// TwinCAT 3 PLC project PLC_Tank
// ProgramVersion: 3.1.4024.0
// libraries:
//   Tc2_ControllerToolbox, * (Beckhoff Automation GmbH)
//   Tc2_ModbusSrv, * (Beckhoff Automation GmbH)
//   Tc2_Standard, * (Beckhoff Automation GmbH)
//   Tc2_System, * (Beckhoff Automation GmbH)
//   Tc3_Module, * (Beckhoff Automation GmbH)
//   VisuDialogs, * (System)
//   VisuSymbols,3.5.10.0,System
// project tree:
//   DUTs/ TAnalogConversion.TcDUT (not stored), TEngine.TcDUT (not stored), TEngineCmd.TcDUT (not stored), THeaterState.TcDUT (not stored), THeaterCmd.TcDUT (not stored), THeater.TcDUT (not stored), TPhaseHeating.TcDUT (not stored), TPhaseCmd.TcDUT (not stored), TPhaseDraining.TcDUT (not stored), TPhaseFilling.TcDUT (not stored), TPhaseMixing.TcDUT (not stored), TPhaseState.TcDUT (not stored), TValveState.TcDUT (not stored), TValveCmd.TcDUT (not stored), TEngineState.TcDUT (not stored), TTank.TcDUT (not stored), TValve.TcDUT (not stored)
//   / GlobalTextList.TcGTLO, PlcTask.TcTTO (not stored), PlcTask500ms.TcTTO (not stored), Visualization Manager.TcVMO (not stored)
//   GVLs/ Global.TcGVL
//   POUs/ Draining.TcPOU, Engine_1DO.TcPOU, FB_Tank.TcPOU (not stored), Filling.TcPOU, Heater.TcPOU, Heating.TcPOU, Main_Batch.TcPOU (not stored), MB_Connector.TcPOU, Mixing.TcPOU, Test.TcPOU (not stored), Valve_2DO.TcPOU, MAIN.TcPOU
//   POUs/Misc/ EngToRaw.TcPOU (not stored), RawToEng.TcPOU (not stored), XNOR.TcPOU
//   VISUs/ Visualization.TcVIS
// real-time tasks:
//   TASK PlcTask: cycle T#100000us, priority 20, ADS port 350
//   TASK PlcTask500ms: cycle T#500ms, priority 1, ADS port 351

// ---- GVLs/Global.TcGVL
{attribute 'qualified_only'}
VAR_GLOBAL
	Tank1 : TTank;
	

	secImp : BOOL;
	
	diMixerRun: BOOL;
	diMixerError : BOOL;
	diValveFillOpen : BOOL;
	diValveFillClose : BOOL;
	diValveFillError : BOOL;
	diValveDrainOpen : BOOL;
	diValveDrainClose : BOOL;
	diValveDrainError : BOOL;
	
	aiWaterLevel : WORD;
	aiWaterTemp : WORD;
	
	doMixerStart : BOOL;
	doValveFillOpen : BOOL;
	doValveFillClose : BOOL;
	doValveDrainOpen : BOOL;
	doValveDrainClose : BOOL;
	doHeatingEnable : BOOL;
	
	aoReqPowerOfHeating : WORD;

END_VAR

VAR_GLOBAL CONSTANT
	Running : INT := 0;
	Stop : INT := 1;
	RunningAndError : INT := 2;
	Err : INT := 3;

	PhIdle : INT := 0;
	PhRunning : INT := 1;
	PhPause : INT := 2;
	
    Open : INT := 0;
	Closed : INT := 1;
	OpenAndErr : INT := 2;
	ClosedAndErr : INT := 3;
	NotOpenNotClosedNotErr : INT := 4;
	NotOpenNotClosedAndErr : INT := 5;
	OpenAndClosedAndErr : INT := 6;
	OpenAndClosedNotErr : INT := 7;
END_VAR

// ---- POUs/Draining.TcPOU
FUNCTION_BLOCK Draining
VAR_INPUT
	diEnabled : BOOL;
END_VAR
VAR_OUTPUT
	doEnabled : BOOL;
END_VAR
VAR_IN_OUT
	DrainingPhase : TPhaseDraining;
	DrainingValve : TValve;
	
END_VAR
VAR
	State_temp	:	INT :=0;
END_VAR

{region "Aut/Man"}
    // switching state of engine - automatic or manual control (default state is manual)
		IF	DrainingPhase.Cmd.ManCtrl	THEN
		DrainingPhase.State.ManCtrl	:= TRUE;
		DrainingPhase.State.AutCtrl := FALSE;			 
	END_IF	 
  
	IF	DrainingPhase.Cmd.AutCtrl	THEN
		DrainingPhase.State.ManCtrl	:= FALSE;
		DrainingPhase.State.AutCtrl := TRUE;			 
	END_IF
		 
	IF	(DrainingPhase.Cmd.ManCtrl AND DrainingPhase.Cmd.AutCtrl) 	THEN
		DrainingPhase.State.ManCtrl	:= TRUE;
		DrainingPhase.State.AutCtrl := FALSE;		 
	END_IF
	
	DrainingPhase.Cmd.ManCtrl	:= FALSE;
	DrainingPhase.Cmd.AutCtrl	:= FALSE;	 
	

{endregion}

{region "ManCtrl"}
    // processing manual actions - if command is processed, it is sets to FALSE even if can't be processed
    // Phase commands are start, stop, pause and resume 
    // Start - open draining valve 
    // Stop - close draining valve
    // Pause - close draining valve
    // Resume - open draining valve
    // real states of phase are writed into states in phase structure
  	IF	DrainingPhase.State.ManCtrl	THEN
			 
	CASE State_temp OF
	
	0:	//IDLE STATE - nothing happens
		 DrainingPhase.State.Running	:= FALSE;
		 DrainingPhase.State.Paused	:= FALSE;
		 DrainingPhase.State.Idle	:= TRUE;
		 IF DrainingPhase.Cmd.StartMan THEN
				  State_temp	:= 1;
			  END_IF
	1:	//RUNNING STATE - manual running
		 DrainingPhase.State.Running	:= TRUE;
		 DrainingPhase.State.Paused	:= FALSE;
		 DrainingPhase.State.Idle	:= FALSE;
		 IF DrainingPhase.Cmd.StopMan THEN
				  State_temp	:= 0;
		 ELSIF DrainingPhase.Cmd.PauseMan THEN
				  State_temp := 2;	
		 	 END_IF
	2:	//PAUSED STATE - in PAUSE you are able to go into either RUNNING or IDLE
		 DrainingPhase.State.Running	:= FALSE;
		 DrainingPhase.State.Paused	:= TRUE;
		 DrainingPhase.State.Idle	:= FALSE;
		IF DrainingPhase.Cmd.ResumeMan THEN
				  State_temp	:= 1;
		 ELSIF DrainingPhase.Cmd.StopMan THEN
				  State_temp := 0;	
		 	END_IF
				  
	END_CASE
		
	DrainingPhase.Cmd.StartMan	:= FALSE; 
	DrainingPhase.Cmd.PauseMan	:= FALSE;
	DrainingPhase.Cmd.StopMan	:= FALSE;
	DrainingPhase.Cmd.ResumeMan	:= FALSE;
   END_IF
	   
{endregion}

{region "AutCtrl"}
    //if request to run in automatic mode -> set auto request to open of filling valve to 1 and close to 0, if not open 0 close 1
    // commands should be sets to false after their processing
	 IF DrainingPhase.State.AutCtrl	THEN
		
	IF	DrainingPhase.Cmd.StartAut THEN
		DrainingPhase.State.Running	:= TRUE;
		DrainingPhase.State.Idle		:= FALSE;	 
	ELSIF	DrainingPhase.Cmd.StopAut THEN	
		DrainingPhase.State.Idle		:= TRUE;
		DrainingPhase.State.Running	:= FALSE;
	END_IF

	DrainingPhase.Cmd.StartAut	:= FALSE;
	DrainingPhase.Cmd.StopAut	:= FALSE;	
   
  END_IF
	
   
{endregion}
{region "Done"}
    //every phase should have finish condition - draining phase - if water level is below requested level
    //after that done state should be setted to 1
   DrainingPhase.ParamDrainLevel	:= 0.02;		//temporary inicialization for testing
		
	IF	DrainingPhase.ParamDrainLevel >= Global.Tank1.Filling.WaterLevel	THEN	//just for now I am using variablbe from Filling	
		DrainingPhase.Cmd.StopMan	:= TRUE;										//perhaps I gotta create new FB EngToRaw for Draining.WaterLevel
		DrainingPhase.Cmd.StopAut	:= TRUE;
		DrainingPhase.State.Done		:= TRUE;		
	ELSIF	DrainingPhase.Cmd.ResetDone THEN
		DrainingPhase.State.Done	:= FALSE;
		DrainingPhase.Cmd.ResetDone := FALSE;
	ELSE
		DrainingPhase.State.Done	:= FALSE;
    END_IF
{endregion}

{region "States"} 
    //Command valve in cases of states
	IF DrainingPhase.State.Running  AND NOT DrainingPhase.State.Idle AND NOT DrainingPhase.State.Paused AND NOT DrainingPhase.State.Done THEN 
        DrainingValve.Cmd.Req2OpenAut := TRUE;
        DrainingValve.Cmd.Req2CloseAut := FALSE;
    ELSE
        DrainingValve.Cmd.Req2OpenAut := FALSE;
        DrainingValve.Cmd.Req2CloseAut := TRUE;
    END_IF;

   
{endregion}

// delault state of phase - if not any state sets state to idle
IF (NOT DrainingPhase.State.Idle) AND (NOT DrainingPhase.State.Paused) AND (NOT DrainingPhase.State.Running) THEN
    DrainingPhase.State.Idle := 1;
END_IF;

// write binary states into int value for visualization
IF DrainingPhase.State.Idle THEN
    DrainingPhase.State.StateInt := Global.PhIdle;
ELSIF DrainingPhase.State.Running THEN
    DrainingPhase.State.StateInt := Global.PhRunning;
ELSE
    DrainingPhase.State.StateInt := Global.PhPause;
END_IF;

//Ponechte pro moznost retezeni volani bloku v LAD
doEnabled := diEnabled;

END_FUNCTION_BLOCK

// ---- POUs/Filling.TcPOU
FUNCTION_BLOCK Filling
VAR_INPUT
	diEnabled : BOOL;
END_VAR
VAR_OUTPUT
	doEnabled : BOOL;
END_VAR
VAR_IN_OUT
	FillingPhase : TPhaseFilling;
	FillingValve : TValve;
END_VAR
VAR
	State_temp	: INT := 0;
END_VAR

{region "REGION Aut/Man"}
    // switching state of engine - automatic or manual control (default state is manual)
	IF	FillingPhase.Cmd.ManCtrl	THEN
		FillingPhase.State.ManCtrl	:= TRUE;
		FillingPhase.State.AutCtrl	:= FALSE;			 
	END_IF	 
  
	IF	FillingPhase.Cmd.AutCtrl	THEN
		FillingPhase.State.ManCtrl	:= FALSE;
		FillingPhase.State.AutCtrl	:= TRUE;			 
	END_IF
		 
	IF	(FillingPhase.Cmd.ManCtrl AND FillingPhase.Cmd.AutCtrl) 	THEN
		FillingPhase.State.ManCtrl	:= TRUE;
		FillingPhase.State.AutCtrl	:= FALSE;			 
	END_IF
	   
	FillingPhase.Cmd.AutCtrl := FALSE;
	FillingPhase.Cmd.ManCtrl := FALSE;
{endregion}

{region "ManCtrl"}
    // processing manual actions - if command is processed, it is sets to FALSE even if can't be processed
    // Phase commands are start, stop, pause and resume 
    // Start - open filling valve 
    // Stop - close filling valve
    // Pause - close filling valve
    // Resume - open filling valve
    // real states of phase are writed into states in phase structure
	
	IF	FillingPhase.State.ManCtrl	THEN
			 
	CASE State_temp OF
	
	0:	//IDLE STATE - nothing happens
		 FillingPhase.State.Running	:= FALSE;
		 FillingPhase.State.Paused	:= FALSE;
		 FillingPhase.State.Idle	:= TRUE;
		 IF FillingPhase.Cmd.StartMan THEN
				  State_temp	:= 1;
			  END_IF
	1:	//RUNNING STATE - manual running
		 FillingPhase.State.Running	:= TRUE;
		 FillingPhase.State.Paused	:= FALSE;
		 FillingPhase.State.Idle	:= FALSE;
		 IF FillingPhase.Cmd.StopMan THEN
				  State_temp	:= 0;
		 ELSIF FillingPhase.Cmd.PauseMan THEN
				  State_temp := 2;	
		 	 END_IF
	2:	//PAUSED STATE - in PAUSE you are able to go into either RUNNING or IDLE
		 FillingPhase.State.Running	:= FALSE;
		 FillingPhase.State.Paused	:= TRUE;
		 FillingPhase.State.Idle	:= FALSE;
		IF FillingPhase.Cmd.ResumeMan THEN
				  State_temp	:= 1;
		 ELSIF FillingPhase.Cmd.StopMan THEN
				  State_temp := 0;	
		 	END_IF
				  
	END_CASE
		
	FillingPhase.Cmd.StartMan	:= FALSE; 
	FillingPhase.Cmd.PauseMan	:= FALSE;
	FillingPhase.Cmd.StopMan	:= FALSE;
	FillingPhase.Cmd.ResumeMan	:= FALSE;
   END_IF
{endregion}

{region "AutCtrl"}
    // if request to run in automatic mode and phase can be run in automatic mode switch phase to running
  IF FillingPhase.State.AutCtrl	THEN
		
	IF	FillingPhase.Cmd.StartAut THEN
		FillingPhase.State.Running	:= TRUE;
		FillingPhase.State.Idle		:= FALSE;	 
	ELSIF	FillingPhase.Cmd.StopAut THEN	
		FillingPhase.State.Idle		:= TRUE;
		FillingPhase.State.Running	:= FALSE;
	END_IF

	FillingPhase.Cmd.StartAut	:= FALSE;
	FillingPhase.Cmd.StopAut	:= FALSE;	
   
  END_IF
			 
   
{endregion}

{region "Done"}
    //every phase should have finish condition - filling phase - if water level is above requested level
    //after that done state should be setted to 1
	FillingPhase.ParamFillLevel	:= 1.5;		//temporary inicialization for testing
		 
	IF	FillingPhase.ParamFillLevel <= FillingPhase.WaterLevel	THEN
		FillingPhase.Cmd.StopMan	:= TRUE;
		FillingPhase.Cmd.StopAut	:= TRUE;
		FillingPhase.State.Done		:= TRUE;		
	ELSIF	FillingPhase.Cmd.ResetDone THEN
		FillingPhase.State.Done	:= FALSE;
		FillingPhase.Cmd.ResetDone := FALSE;
    END_IF
{endregion}

{region "States"} 
    //Command valve in cases of states
	IF FillingPhase.State.Running  AND NOT FillingPhase.State.Idle AND NOT FillingPhase.State.Paused AND NOT FillingPhase.State.Done THEN 
        FillingValve.Cmd.Req2OpenAut := TRUE;
		FillingValve.Cmd.Req2CloseAut := FALSE;			 
    ELSE
        FillingValve.Cmd.Req2OpenAut := FALSE;
        FillingValve.Cmd.Req2CloseAut := TRUE;
    END_IF;

{endregion}


// delault state of phase - if not any state sets state to idle
IF NOT FillingPhase.State.Idle AND NOT FillingPhase.State.Paused AND NOT FillingPhase.State.Running THEN
    FillingPhase.State.Idle := 1;
END_IF;

// write binary states into int value for visualization
IF FillingPhase.State.Idle THEN
    FillingPhase.State.Stateint := Global.PhIdle;
ELSIF FillingPhase.State.Running THEN
    FillingPhase.State.Stateint := Global.PhRunning;
ELSE
    FillingPhase.State.Stateint := Global.PhPause;
END_IF;

// Ponechte pro moznost retezeni volani bloku v LAD
doEnabled := diEnabled;

END_FUNCTION_BLOCK

// ---- POUs/Engine_1DO.TcPOU
FUNCTION_BLOCK Engine_1DO
VAR_INPUT
	iRunning : BOOL;
	iError : BOOL;
	iSecImp : BOOL;
END_VAR
VAR_OUTPUT
	oRun : BOOL;
END_VAR
VAR_IN_OUT
	ioEngStruct : TEngine;
END_VAR
VAR
	secImpEdge: BOOL;
	tempStartupFail: BOOL;
END_VAR

{region "RunState"}
    // set real state of engine run into engine structure
		 
 ioEngStruct.State.Run := iRunning;

{endregion}

{region "Running time"} 
    // counting running time of engine - (motoseconds in real situation it should be moto hours)
    // detection rising edge of input secimp - should be conected 1Hz internal clock from PLC
		 
			  
	
{endregion}
	 
 
{region "Manual/Automat"}
	// switching state of engine - automatic or manual control (default state is manual)
	IF ioEngStruct.Cmd.ManCtrl	THEN
		ioEngStruct.State.ManCtrl	:= TRUE;
		ioEngStruct.State.AutCtrl	:= FALSE;
	ELSIF	ioEngStruct.Cmd.AutCtrl	THEN
		ioEngStruct.State.ManCtrl	:= FALSE;
		ioEngStruct.State.AutCtrl	:= TRUE;
	ELSIF	XNOR(A := ioEngStruct.Cmd.AutCtrl,B := ioEngStruct.Cmd.ManCtrl ) THEN
		ioEngStruct.State.ManCtrl	:= TRUE;
		ioEngStruct.State.AutCtrl	:= FALSE;		
	END_IF 
	ioEngStruct.State.ManCtrl	:= FALSE;
	ioEngStruct.State.AutCtrl	:= FALSE;
	
{endregion}
	 
{region "MayRun / MayAutoRun"}
	// setting auxilary signals (may run, may auto run) - MR AND NOT MAR - eng should be started in manual mode,
    // MAR - should be started in automatic mode
    ioEngStruct.State.MayRun := (ioEngStruct.State.ManCtrl AND NOT(ioEngStruct.State.GenErr));
	ioEngStruct.State.MayAutoRun := (ioEngStruct.State.AutCtrl AND NOT(ioEngStruct.State.GenErr));
		 
			  
{endregion}
	 
{region "ManCtrl"}
	// processing manual actions - if command is processed, it is set to FALSE even if can't be processed
    // Engine commands are turn off (stop) and turn on (start)
	
{endregion}
	 
{region "AutCtrl"}
	//if request to run in automatic mode set outputs to right states if MAR
    //AutoRequest shouldn't be reseted to false state
    
{endregion}
	 
{region "Error states"}
	// definition of error states 
	// error - input from digital input of plc - fyzical state of engine 
	// calculating start up fail - if output is sets to start engine, it's expected feedback from running signal in defined time, if feedback doesn't show in this time, it should be start up fail error
	// merge of these two error is general error
	
{endregion}
	 
oRun := ioEngStruct.State.RunOut;

{region "StatusInt"}
 IF NOT ioEngStruct.State.GenErr THEN
        IF ioEngStruct.State.Run THEN
            ioEngStruct.State.StateInt := Global.Running;
        ELSE
            ioEngStruct.State.StateInt := Global.Stop;
        END_IF;
    ELSE
        IF ioEngStruct.State.Run THEN
            ioEngStruct.State.StateInt := Global.RunningAndError;
        ELSE
            ioEngStruct.State.StateInt := Global.Err;
        END_IF;
    END_IF; 
{endregion}

END_FUNCTION_BLOCK

// ---- POUs/Misc/XNOR.TcPOU
FUNCTION XNOR : BOOL
VAR_INPUT
	A	:	BOOL;
	B	:	BOOL;
END_VAR
VAR
END_VAR

XNOR := (A AND B) OR ((NOT A) AND  (NOT B));

END_FUNCTION

// ---- POUs/Heater.TcPOU
FUNCTION_BLOCK Heater
VAR_INPUT
	iWaterTemp : REAL;
END_VAR
VAR_OUTPUT
	oHeaterEnable : BOOL;
	oHeaterPower : REAL;
END_VAR
VAR_IN_OUT
	ioHeatStruct : THeater;
END_VAR
VAR
	pidParameters : ST_CTRL_PID_PARAMS;
END_VAR

pidParameters.fKp := 10; //P
pidParameters.tTn := T#2S; //I
pidParameters.tTv := T#0.5S; //D
pidParameters.tCtrlCycleTime := T#200MS;
pidParameters.tTaskCycleTime := T#100MS;
pidParameters.fOutMaxLimit := 100;
pidParameters.fOutMinLimit := 0;
pidParameters.bDInTheFeedbackPath := FALSE;
pidParameters.bPInTheFeedbackPath := FALSE;
pidParameters.bARWOnIPartOnly := FALSE;
pidParameters.tTd := T#100MS; 

ioHeatStruct.PID(
	fSetpointValue := ioHeatStruct.ParamHeatingSetPointAutomat, 
	fActualValue := iWaterTemp, 
	fManSyncValue := ioHeatStruct.ParamHeatingPowerManual,
	bSync := ioHeatStruct.State.ManCtrl,
	eMode := E_CTRL_MODE.eCTRL_MODE_ACTIVE, // automatic mode of PID component
	stParams := pidParameters);

ioHeatStruct.State.HeatingOut := ioHeatStruct.PID.fOut;

	 
{region "Manual/Automat"}
// switching state of engine - automatic or manual control (default state is manual)
	IF ioHeatStruct.Cmd.ManCtrl OR ioHeatStruct.State.GenErr THEN 
		ioHeatStruct.State.ManCtrl := TRUE;	  
		ioHeatStruct.State.AutCtrl := FALSE;
	END_IF
		 
	IF ioHeatStruct.Cmd.AutCtrl  AND NOT ioHeatStruct.Cmd.ManCtrl AND NOT ioHeatStruct.State.GenErr THEN
		ioHeatStruct.State.AutCtrl := TRUE;	 
		ioHeatStruct.State.ManCtrl := FALSE; 
	END_IF
		 
	IF  ioHeatStruct.State.AutCtrl  = ioHeatStruct.State.ManCtrl THEN 
		ioHeatStruct.State.AutCtrl := FALSE;	 
		ioHeatStruct.State.ManCtrl := TRUE; 
	END_IF
		 
	ioHeatStruct.Cmd.ManCtrl := FALSE;
	ioHeatStruct.Cmd.AutCtrl := FALSE;

{endregion}
	 
 
{region "ManCtrl"}
// processing manual actions - if command is processed, it is set to FALSE even if can't be processed
// Engine commands are turn off (stop) and turn on (start)
IF ioHeatStruct.State.ManCtrl  	THEN
	
	IF ioHeatStruct.Cmd.TurnOnMan	THEN
		ioHeatStruct.State.EnableOut	:= TRUE;
		END_IF	
	IF	ioHeatStruct.Cmd.TurnOffMan	THEN
		ioHeatStruct.State.EnableOut	:= FALSE;
		END_IF	
	IF	ioHeatStruct.Cmd.TurnOffMan =  ioHeatStruct.Cmd.TurnOnMan	THEN
		ioHeatStruct.State.EnableOut	:= FALSE;
		END_IF	
						   
END_IF
		

{endregion}
 
{region "AutCtrl"}
//if request to run in automatic mode set outputs to right states if MAR
//AutoRequest shouldn't be reseted to false state

{endregion}
 
{region "Error states"}
ioHeatStruct.ParamHeatingSetPointAutomat	:= 90;
{endregion}
// if water temperature is too high, stop heating and generate error
	IF iWaterTemp > ioHeatStruct.ParamHeatingSetPointAutomat THEN
		ioHeatStruct.State.Err := TRUE;
		oHeaterEnable := FALSE;
	END_IF
	 
{endregion}
	 
 
oHeaterPower := ioHeatStruct.State.HeatingOut;
oHeaterEnable := ioHeatStruct.State.EnableOut;

END_FUNCTION_BLOCK

// ---- POUs/Heating.TcPOU
FUNCTION_BLOCK Heating
VAR_INPUT
	diEnabled : BOOL;
	iSecImp : BOOL;
END_VAR
VAR_OUTPUT
	doEnabled : BOOL;
END_VAR
VAR_IN_OUT
	HeatingPhase : TPhaseHeating;
	Heater : THeater;
END_VAR
VAR
	pidParameters : ST_CTRL_PID_PARAMS;
END_VAR


{region "Aut/Man"}
    // switching state of engine - automatic or manual control (default state is manual)
 
{endregion}

{region "ManCtrl"}
    // processing manual actions - if command is processed, it is sets to FALSE even if can't be processed
        // real states of phase are writed into states in phase structure
    
   
{endregion}

{region "AutCtrl"}
    // if request to run in automatic mode -> set auto request to heat to 1, if not request to heat 0
    // commands should be sets to false after their processing
  
{endregion}

{region "Done"}
    //every phase should have finish condition - heating phase - if water temp is on requested value for 15 seconds with 1°C hysteresis
    //after that done state should be setted to 1



    // command reset done resets done state and than resets command
  
{endregion}

{region "States"}
    //Command valve in cases of states
    // Running - start heating  
    // Idle - stop heating
    // Pause - stop heating (alternative is hold actual temp)
  
{endregion}

// delault state of phase - if not any state sets state to idle
IF NOT HeatingPhase.State.Idle AND NOT HeatingPhase.State.Paused AND NOT HeatingPhase.State.Running THEN
    HeatingPhase.State.Idle := 1;
END_IF;

doEnabled := diEnabled;

END_FUNCTION_BLOCK

// ---- POUs/MB_Connector.TcPOU
PROGRAM MB_Connector
VAR
	
	mb_ipaddr   : STRING(15) := '127.0.0.1';
	mb_port		: UINT := 503;
	mb_unitid	: BYTE := 1;
	
	fbReadRegs		: FB_MBReadInputRegs;
	mb_regs    		: ARRAY [0..4] OF WORD;
	mb_regs_error	: BOOL;
	mb_regs_busy	: BOOL;
	mb_regs_execute : BOOL;
	mb_regs_errid	: UDINT;
	
	fbReadInps	: FB_MBReadInputs;
	mb_inps			: ARRAY [0..4] OF BYTE;
	mb_inps_error	: BOOL;
	mb_inps_busy	: BOOL;
	mb_inps_execute : BOOL;
	mb_inps_errid	: UDINT;
	
	fbWriteRegs		: FB_MBWriteRegs;
	mbw_regs    	: ARRAY [0..4] OF WORD;
	mbw_regs_error	: BOOL;
	mbw_regs_busy	: BOOL;
	mbw_regs_execute: BOOL;
	mbw_regs_errid	: UDINT;
	
	fbWriteCoils	: FB_MBWriteCoils;
	mbw_coils		: ARRAY [0..4] OF BYTE;
	mbw_coils_error	: BOOL;
	mbw_coils_busy	: BOOL;
	mbw_coils_execute: BOOL;
	mbw_coils_errid	: UDINT;
	
END_VAR

fbReadRegs.sIPAddr := mb_ipaddr;
fbReadRegs.nTCPPort := mb_port;
fbReadRegs.nQuantity := 4;
fbReadRegs.nMBAddr := 0;
fbReadRegs.cbLength := SIZEOF(mb_regs);
fbReadRegs.pDestAddr := ADR(mb_regs);
fbReadRegs.nUnitID := mb_unitid;
fbReadRegs.tTimeout := T#5S;
IF (mb_regs_busy = FALSE) THEN
	mb_regs_execute := TRUE;
ELSE
	mb_regs_execute := FALSE;
END_IF
fbReadRegs(bExecute := mb_regs_execute, 
		   bBusy => mb_regs_busy, bError => mb_regs_error, 
		   nErrId => mb_regs_errid);



fbReadInps.sIPAddr := mb_ipaddr;
fbReadInps.nTCPPort := mb_port;
fbReadInps.nQuantity := 32;
fbReadInps.nMBAddr := 0;
fbReadInps.cbLength := SIZEOF(mb_inps);
fbReadInps.pDestAddr := ADR(mb_inps);
fbReadInps.nUnitID := mb_unitid;
fbReadInps.tTimeout := T#5S;
IF (mb_inps_busy = FALSE) THEN
	
	mb_inps_execute := TRUE;
ELSE
	mb_inps_execute := FALSE;
END_IF
fbReadInps(bExecute := mb_inps_execute, 
	bBusy => mb_inps_busy, bError => mb_inps_error, nErrId => mb_inps_errid);
Global.diValveFillOpen := mb_inps[0].0;
Global.diValveFillClose := mb_inps[0].1;
Global.diValveFillError := mb_inps[0].2;
Global.diValveDrainOpen := mb_inps[0].3;
Global.diValveDrainClose := mb_inps[0].4;
Global.diValveDrainError := mb_inps[0].5;
Global.diMixerRun := mb_inps[0].6;
Global.diMixerError := mb_inps[0].7;

Global.aiWaterLevel := mb_regs[0];
Global.aiWaterTemp := mb_regs[2];







fbWriteRegs.sIPAddr := mb_ipaddr;
fbWriteRegs.nTCPPort := mb_port;
fbWriteRegs.nQuantity := 4;
fbWriteRegs.nMBAddr := 0;
fbWriteRegs.cbLength := SIZEOF(mbw_regs);
fbWriteRegs.pSrcAddr := ADR(mbw_regs);
fbWriteRegs.nUnitID := mb_unitid;
fbWriteRegs.tTimeout := T#5S;
IF (mbw_regs_busy = FALSE) THEN
	mbw_regs_execute := TRUE;
ELSE
	mbw_regs_execute := FALSE;
END_IF
fbWriteRegs(bExecute := mbw_regs_execute, 
		   bBusy => mbw_regs_busy, bError => mbw_regs_error, 
		   nErrId => mbw_regs_errid);



fbWriteCoils.sIPAddr := mb_ipaddr;
fbWriteCoils.nTCPPort := mb_port;
fbWriteCoils.nQuantity := 32;
fbWriteCoils.nMBAddr := 0;
fbWriteCoils.cbLength := SIZEOF(mbw_coils);
fbWriteCoils.pSrcAddr := ADR(mbw_coils);
fbWriteCoils.nUnitID := mb_unitid;
fbWriteCoils.tTimeout := T#5S;
IF (mbw_coils_busy = FALSE) THEN
	mbw_coils_execute := TRUE;
ELSE
	mbw_coils_execute := FALSE;
END_IF
fbWriteCoils(bExecute := mbw_coils_execute, 
	bBusy => mbw_coils_busy, bError => mbw_coils_error, nErrId => mbw_coils_errid);

mbw_coils[0].0 := Global.doValveFillOpen;
mbw_coils[0].1 := Global.doValveFillClose;
mbw_coils[0].2 := Global.doValveDrainOpen;
mbw_coils[0].3 := Global.doValveDrainClose;
mbw_coils[0].4 := Global.doMixerStart;
mbw_coils[0].5 := Global.doHeatingEnable;

mbw_regs[0] := Global.aoReqPowerOfHeating;

END_PROGRAM

// ---- POUs/Mixing.TcPOU
FUNCTION_BLOCK Mixing
VAR_INPUT
	diEnabled : BOOL;
	iSecImp : BOOL;
END_VAR
VAR_OUTPUT
	doEnabled : BOOL;
END_VAR
VAR_IN_OUT
	MixingPhase : TPhaseMixing;
	MixerEng : TEngine;
END_VAR
VAR
END_VAR

{region "Aut/Man"}
    // switching state of engine - automatic or manual control (default state is manual)
  
{endregion}

{region "ManCtrl"}
    // processing manual actions - if command is processed, it is sets to FALSE even if can't be processed
    // Phase commands are start, stop, pause and resume 
    // Start - start mixing  
    // Stop - stop mixing
    // Pause - stop mixing 
    // Resume - start mixing
    // real states of phase are writed into states in phase structure
   
{endregion}

{region "AutCtrl"}
    // if request to run in automatic mode -> set auto request to mixing to 1, if not request to mixing is 0
    // commands should be sets to false after their processing
   
{endregion}

{region "Done"}
    // every phase should have finish condition - mixing phase - if time of runnig is bigger or same as requested
    // after that done state should be setted to 1
 
{endregion}

{region "States"}
    //Command mixer in cases of states

{endregion}


// delault state of phase - if not any state sets state to idle
IF NOT MixingPhase.State.Idle AND NOT MixingPhase.State.Done AND NOT MixingPhase.State.Paused AND NOT MixingPhase.State.Running THEN
    MixingPhase.State.Idle := 1;
END_IF;


// delault state of phase - if not any state sets state to idle
IF MixingPhase.State.Idle THEN
    MixingPhase.State.StateInt := Global.PhIdle;
ELSIF MixingPhase.State.Running THEN
    MixingPhase.State.StateInt := Global.PhRunning;
ELSE
    MixingPhase.State.StateInt := Global.PhPause;
END_IF;

doEnabled := diEnabled;

END_FUNCTION_BLOCK

// ---- POUs/Valve_2DO.TcPOU
FUNCTION_BLOCK Valve_2DO
VAR_INPUT
	iOpen : BOOL;
	iClose : BOOL;
	iError : BOOL;
	iSecImp : BOOL;
END_VAR
VAR_OUTPUT
	oOpen : BOOL;
	oClose : BOOL;
END_VAR

VAR_IN_OUT
	ioValStruct	 : TValve;
END_VAR

VAR
	tempOpenStartupFail : BOOL;
	tempCloseStartupFail: BOOL;
END_VAR

{region "OpenState"}
    // set real state of valve input into valve structure - input of valve can be taken from limit sensor...
    ioValStruct.State.Open := iOpen;
    ioValStruct.State.Closed := iClose;
{endregion}

	 
{region "Manual/Automat"}
	// switching state of engine - automatic or manual control (default state is manual)
		 IF ioValStruct.Cmd.ManCtrl THEN
			ioValStruct.State.ManCtrl := TRUE;
			ioValStruct.State.AutCtrl :=FALSE;				 					  
		 END_IF
			  
		 IF ioValStruct.State.GenErr THEN
			ioValStruct.State.ManCtrl := TRUE;
			ioValStruct.State.AutCtrl :=FALSE;
		 END_IF
				 
	
		 IF ioValStruct.Cmd.AutCtrl THEN
			ioValStruct.State.ManCtrl := FALSE;
		    ioValStruct.State.AutCtrl := TRUE;					   
		 END_IF
			  
		IF (ioValStruct.Cmd.ManCtrl AND ioValStruct.Cmd.AutCtrl)	THEN
			ioValStruct.State.ManCtrl	:= TRUE;
			ioValStruct.State.AutCtrl	:= FALSE; 
		END_IF

    ioValStruct.Cmd.ManCtrl := FALSE;
    ioValStruct.Cmd.AutCtrl := FALSE;	
	
{endregion}
	
{region "MayRun / MayAutoRun"}
    // setting auxilary signals (may run, may auto run) - MR AND NOT MAR - engine may be started in manual mode, MAR - engine may be started in automatic mode
    ioValStruct.State.MayRun := (ioValStruct.State.ManCtrl AND NOT(ioValStruct.State.GenErr));
	ioValStruct.State.MayAutoRun := (ioValStruct.State.AutCtrl AND NOT(ioValStruct.State.GenErr));
{endregion}
	 
{region "ManCtrl"}
	// processing manual actions - if command is processed, it is sets to FALSE even if can't be processed
    // Valve commands are open, close and stop - valve can be stopped intermediate position
	 IF ioValStruct.State.ManCtrl AND ioValStruct.State.MayRun THEN
        IF ioValStruct.Cmd.OpenMan THEN
            ioValStruct.State.CloseOut := FALSE;
            ioValStruct.State.OpenOut := TRUE;
        END_IF;
        
        IF ioValStruct.Cmd.CloseMan THEN
            ioValStruct.State.OpenOut := FALSE;
            ioValStruct.State.CloseOut := TRUE;
        END_IF;
        
        IF ioValStruct.Cmd.StopMan THEN
            ioValStruct.State.OpenOut := FALSE;
            ioValStruct.State.CloseOut := TRUE;
        END_IF;
    END_IF;
    
    ioValStruct.Cmd.OpenMan := FALSE;
    ioValStruct.Cmd.CloseMan := FALSE;
    ioValStruct.Cmd.StopMan := FALSE;
{endregion}
	 
{region "AutCtrl"}
	 //if request to run in automatic mode -> set outputs to right states if MAR
    //AutoRequest shouldn't be reseted to false state
    //if request to open and request to close are setted to 1 simultaneously - outputs should be 0.
    IF ioValStruct.State.AutCtrl AND ioValStruct.State.MayAutoRun THEN
        IF ioValStruct.Cmd.Req2CloseAut AND (NOT ioValStruct.Cmd.Req2OpenAut) THEN
            ioValStruct.State.OpenOut := FALSE;
            ioValStruct.State.CloseOut := TRUE;
        END_IF;
        
        IF (NOT ioValStruct.Cmd.Req2CloseAut) AND ioValStruct.Cmd.Req2OpenAut THEN
            ioValStruct.State.CloseOut := FALSE;
            ioValStruct.State.OpenOut := TRUE;
        END_IF;
        
        IF (NOT ioValStruct.Cmd.Req2CloseAut) AND (NOT ioValStruct.Cmd.Req2OpenAut) THEN
            ioValStruct.State.CloseOut := FALSE;
            ioValStruct.State.OpenOut := FALSE;
        END_IF;
        
    END_IF;
{endregion}
	 
{region "Error states"}
 // definition of error states 
    // error - input from digital input of plc - fyzical state of valve
    // calculating start up fail - if output is sets to open or close, it's expected feedback from limit sensor in defined time, if feedback doesn't show in this time, it should be start up fail error
    // merge of these two error is general error
    // error is both inputs (open and closed) true state
    ioValStruct.OpenFailTimer(IN := (ioValStruct.State.OpenOut AND (NOT ioValStruct.State.CloseOut)), PT := ioValStruct.Time2Open);
	IF	ioValStruct.OpenFailTimer.Q AND NOT ioValStruct.State.Open	THEN	//MANDATORY CONDITION (I had to add Input from sensor)
		tempOpenStartupFail := TRUE;								
	END_IF

    ioValStruct.CloseFailTimer(IN := ((NOT ioValStruct.State.OpenOut) AND ioValStruct.State.CloseOut), PT := ioValStruct.Time2Open);
	IF	ioValStruct.OpenFailTimer.Q AND NOT ioValStruct.State.Open	THEN	//MANDATORY CONDITION (I had to add Input from sensor)
		tempCloseStartupFail := TRUE;							
	END_IF	

    
   
    IF tempOpenStartupFail OR tempCloseStartupFail THEN
        ioValStruct.State.StartUpFail := TRUE;
    END_IF;
    
    IF iError THEN
        ioValStruct.State.Err := TRUE;
    END_IF;
    
    ioValStruct.State.GenErr := ioValStruct.State.StartUpFail OR iError;
    
    // start up fail can be reseted by operator, command resetSUF, resets SUF and engine should be started again
    IF ioValStruct.Cmd.ResetSUF THEN
        ioValStruct.State.StartUpFail := FALSE;
        ioValStruct.Cmd.ResetSUF := FALSE;
    END_IF;
    
    // if error state exists outputs should be in stop state
    IF ioValStruct.State.GenErr THEN
        ioValStruct.State.OpenOut := FALSE;
        ioValStruct.State.CloseOut := FALSE;
    END_IF;
{endregion}
	 	 
oOpen := ioValStruct.State.OpenOut;
oClose := ioValStruct.State.CloseOut;

{region "StatusInt"}
    //write combination of states into int value for visualization (valve - combination of open, close state and error)
    IF ioValStruct.State.Open AND NOT ioValStruct.State.Closed AND NOT ioValStruct.State.GenErr THEN
        ioValStruct.State.StColor := Global.Open;
    ELSIF NOT ioValStruct.State.Open AND ioValStruct.State.Closed AND NOT ioValStruct.State.GenErr THEN
        ioValStruct.State.StColor := Global.Closed;
    ELSIF ioValStruct.State.Open AND NOT ioValStruct.State.Closed AND ioValStruct.State.GenErr THEN
        ioValStruct.State.StColor := Global.OpenAndErr;
    ELSIF NOT ioValStruct.State.Open AND ioValStruct.State.Closed AND ioValStruct.State.GenErr THEN
        ioValStruct.State.StColor := Global.ClosedAndErr;
    ELSIF NOT ioValStruct.State.Open AND NOT ioValStruct.State.Closed AND NOT ioValStruct.State.GenErr THEN
        ioValStruct.State.StColor := Global.NotOpenNotClosedNotErr;
    ELSIF NOT ioValStruct.State.Open AND NOT ioValStruct.State.Closed AND ioValStruct.State.GenErr THEN
        ioValStruct.State.StColor := Global.NotOpenNotClosedAndErr;
    ELSIF ioValStruct.State.Open AND ioValStruct.State.Closed AND ioValStruct.State.GenErr THEN
        ioValStruct.State.StColor := Global.OpenAndClosedAndErr;
    ELSIF ioValStruct.State.Open AND ioValStruct.State.Closed AND NOT ioValStruct.State.GenErr THEN
        ioValStruct.State.StColor := Global.OpenAndClosedNotErr;
    END_IF;
{endregion}

END_FUNCTION_BLOCK

// ---- POUs/MAIN.TcPOU
PROGRAM MAIN
VAR

END_VAR

Global.secImp := NOT(Global.secImp);

END_PROGRAM

// ---- GlobalTextList.TcGTLO
TEXTLIST GlobalTextList
  815 = 'ABC'
  406 = 'AUT'
  736 = 'AUTOMAT'
  322 = 'Automat'
  473 = 'Checkbox'
  70 = 'Close'
  25 = 'Closed'
  655 = 'Done'
  220 = 'DRAIN - Control moudule (CM)'
  110 = 'DRAIN - PHASE'
  177 = 'FILL - Control moudule (CM)'
  836 = 'FILL - PHASE'
  296 = 'FILL- Control moudule (CM)'
  18 = 'FILL- Valve Control moudule (CM)'
  960 = 'Filling phase'
  211 = 'Filling States'
  557 = 'Filling states'
  201 = 'Filling Valve'
  558 = 'Idle'
  560 = 'MAN'
  854 = 'MANUAL'
  397 = 'Manual'
  57 = 'Mixer- Control moudule (CM)'
  604 = 'Open'
  687 = 'Opened'
  435 = 'Pause'
  750 = 'PAUSE'
  487 = 'Paused'
  98 = 'Res. SUF'
  478 = 'Reset done'
  742 = 'RESUME'
  331 = 'Running'
  400 = 'START'
  884 = 'STOP'
  256 = 'SUF'
  415 = 'VALVE - Control moudule (CM)'
  780 = 'VALVE Control moudule (CM)'
END_TEXTLIST

// ---- VISUs/Visualization.TcVIS
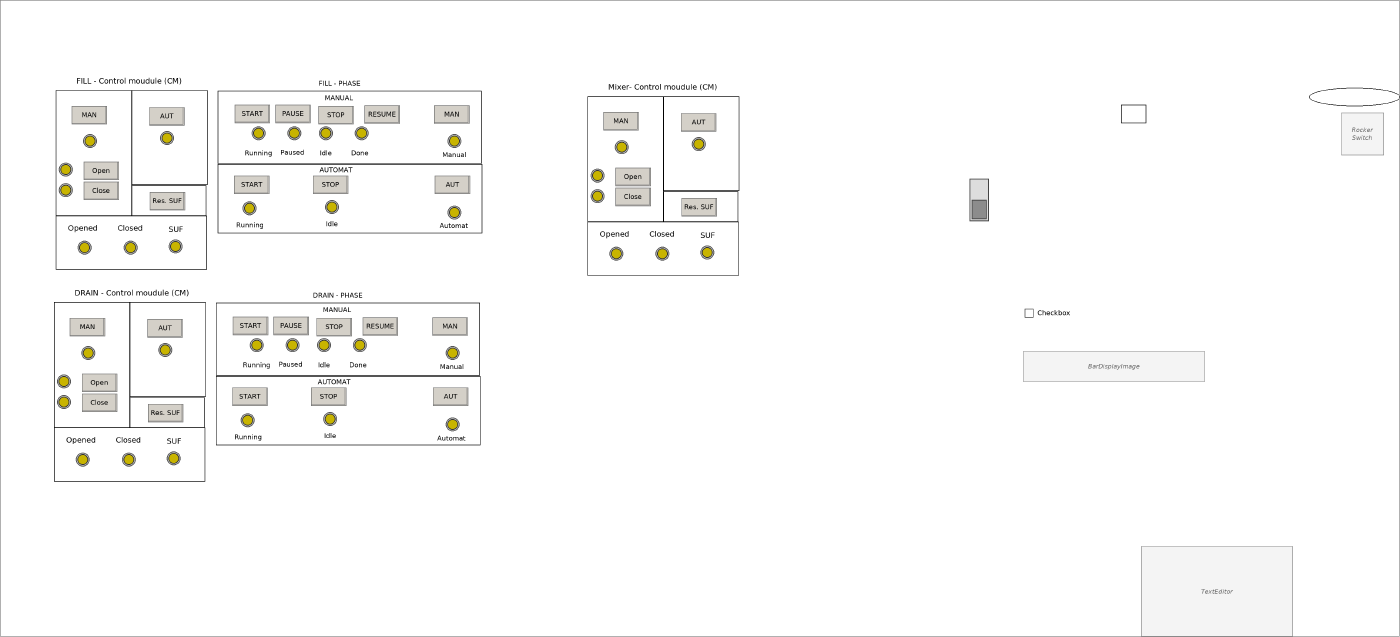
VISUALIZATION Visualization  // 2309x1052
    Rectangle (217,149 125x156)
    Rectangle (217,306 123x50)
    Rectangle (92,149 125x207)
    Rectangle (359,271 436x114)
    Rectangle (92,356 249x89)
    Checkbox (1688,502 150x30), "Checkbox"
    BarDisplayImage (1687,580 300x50), style: BarDisplayImage-Gray, scale format: %.1f, scale 0..100
    DipSwitch (1580,295 70x70), behaviour: TOGGLE, style: Switch-DipSwitch-Gray
    RockerSwitch (2212,186 70x70), behaviour: TOGGLE, style: Switch-RockerSwitch-Gray
    TextEditor (1882,902 250x150)
        p4127561890: Courier New
    Ellipse (2159,145 150x30)
    Rectangle (1849,173 41x30)
    Button (246,177 58x30), "AUT"
        OnMouseClick: toggle Global.Tank1.ValveFilling.Cmd.AutCtrl
    Button (118,175 58x30), "MAN"
        OnMouseClick: toggle Global.Tank1.ValveFilling.Cmd.ManCtrl
    Label (123,125 212x18), "FILL - Control moudule (CM)"
    Button (138,267 58x30), "Open"
        OnMouseClick: toggle Global.Tank1.ValveFilling.Cmd.OpenMan
    Button (138,300 58x30), "Close"
        OnMouseClick: toggle Global.Tank1.ValveFilling.Cmd.CloseMan
    Lamp1 (262,215 27x26), variable: Global.Tank1.ValveFilling.State.AutCtrl, style: Lamp-Lamp1-Yellow
    Lamp1 (135,220 27x26), variable: Global.Tank1.ValveFilling.State.ManCtrl, style: Lamp-Lamp1-Yellow
    Lamp1 (126,396 27x26), variable: Global.Tank1.ValveFilling.State.Open, style: Lamp-Lamp1-Yellow
    Lamp1 (202,396 27x26), variable: Global.Tank1.ValveFilling.State.Closed, style: Lamp-Lamp1-Yellow
    Lamp1 (276,394 27x26), variable: Global.Tank1.ValveFilling.State.StartupFail, style: Lamp-Lamp1-Yellow
    Button (247,317 58x30), "Res. SUF"
        OnMouseClick: toggle Global.Tank1.ValveFilling.Cmd.ResetSUF
    Label (109,368 53x18), "Opened"
    Label (191,368 53x18), "Closed"
    Label (275,370 33x18), "SUF"
    Lamp1 (95,267 27x26), variable: Global.Tank1.ValveFilling.State.OpenOut, style: Lamp-Lamp1-Yellow
    Lamp1 (95,301 27x26), variable: Global.Tank1.ValveFilling.State.CloseOut, style: Lamp-Lamp1-Yellow
    Rectangle (359,150 435x120)
    Lamp1 (413,207 27x26), variable: Main_Batch.FB_Tank_1.FillingPhase.FillingPhase.State.Running, style: Lamp-Lamp1-Yellow
    Lamp1 (472,207 27x26), variable: Global.Tank1.Filling.State.Paused, style: Lamp-Lamp1-Yellow
    Lamp1 (524,207 27x26), variable: Global.Tank1.Filling.State.Idle, style: Lamp-Lamp1-Yellow
    Lamp1 (583,207 27x26), variable: Global.Tank1.Filling.State.Done, style: Lamp-Lamp1-Yellow
    Label (485,123 150x30), "FILL - PHASE"
    Label (400,238 53x30), "Running"
    Label (456,237 53x30), "Paused"
    Label (511,238 53x30), "Idle"
    Label (567,238 53x30), "Done"
    Button (717,290 58x30), "AUT"
        OnMouseClick: toggle Global.Tank1.Filling.Cmd.AutCtrl
    Button (716,174 58x30), "MAN"
        OnMouseClick: toggle Global.Tank1.Filling.Cmd.ManCtrl
    Lamp1 (736,338 27x26), variable: Global.Tank1.Filling.State.AutCtrl, style: Lamp-Lamp1-Yellow
    Lamp1 (736,220 27x26), variable: Global.Tank1.Filling.State.ManCtrl, style: Lamp-Lamp1-Yellow
    Button (387,173 58x30), "START"
        OnMouseClick: toggle Global.Tank1.Filling.Cmd.StartMan
    Button (454,173 58x30), "PAUSE"
        OnMouseClick: toggle Global.Tank1.Filling.Cmd.PauseMan
    Button (525,175 58x30), "STOP"
        OnMouseClick: toggle Global.Tank1.Filling.Cmd.StopMan
    Button (601,174 58x30), "RESUME"
        OnMouseClick: toggle Global.Tank1.Filling.Cmd.ResumeMan
    Button (386,290 58x30), "START"
        OnMouseClick: toggle Global.Tank1.Filling.Cmd.StartAut
    Button (516,290 58x30), "STOP"
        OnMouseClick: toggle Global.Tank1.Filling.Cmd.StopAut
    Lamp1 (398,331 27x26), variable: Global.Tank1.Filling.State.Running, style: Lamp-Lamp1-Yellow
    Lamp1 (534,329 27x26), variable: Global.Tank1.Filling.State.Idle, style: Lamp-Lamp1-Yellow
    Label (484,147 150x30), "MANUAL"
    Label (479,266 150x30), "AUTOMAT"
    Label (386,357 53x30), "Running"
    Label (521,355 53x30), "Idle"
    Rectangle (214,499 125x156)
    Rectangle (214,656 123x50)
    Rectangle (89,499 125x207)
    Rectangle (356,621 436x114)
    Rectangle (89,706 249x89)
    Button (243,527 58x30), "AUT"
        OnMouseClick: toggle Global.Tank1.ValveDraining.Cmd.AutCtrl
    Button (115,525 58x30), "MAN"
        OnMouseClick: toggle Global.Tank1.ValveDraining.Cmd.ManCtrl
    Label (120,475 212x18), "DRAIN - Control moudule (CM)"
    Button (135,617 58x30), "Open"
        OnMouseClick: toggle Global.Tank1.ValveDraining.Cmd.OpenMan
    Button (135,650 58x30), "Close"
        OnMouseClick: toggle Global.Tank1.ValveDraining.Cmd.CloseMan
    Lamp1 (259,565 27x26), variable: Global.Tank1.ValveDraining.State.AutCtrl, style: Lamp-Lamp1-Yellow
    Lamp1 (132,570 27x26), variable: Global.Tank1.ValveDraining.State.ManCtrl, style: Lamp-Lamp1-Yellow
    Lamp1 (123,746 27x26), variable: Global.Tank1.ValveFilling.State.Open, style: Lamp-Lamp1-Yellow
    Lamp1 (199,746 27x26), variable: Global.Tank1.ValveFilling.State.Closed, style: Lamp-Lamp1-Yellow
    Lamp1 (273,744 27x26), variable: Global.Tank1.ValveDraining.State.StartupFail, style: Lamp-Lamp1-Yellow
    Button (244,667 58x30), "Res. SUF"
        OnMouseClick: toggle Global.Tank1.ValveDraining.Cmd.ResetSUF
    Label (106,718 53x18), "Opened"
    Label (188,718 53x18), "Closed"
    Label (272,720 33x18), "SUF"
    Lamp1 (92,617 27x26), variable: Global.Tank1.ValveDraining.State.OpenOut, style: Lamp-Lamp1-Yellow
    Lamp1 (92,651 27x26), variable: Global.Tank1.ValveDraining.State.CloseOut, style: Lamp-Lamp1-Yellow
    Rectangle (356,500 435x120)
    Lamp1 (410,557 27x26), variable: Global.Tank1.Draining.State.Running, style: Lamp-Lamp1-Yellow
    Lamp1 (469,557 27x26), variable: Global.Tank1.Draining.State.Paused, style: Lamp-Lamp1-Yellow
    Lamp1 (521,557 27x26), variable: Global.Tank1.Draining.State.Idle, style: Lamp-Lamp1-Yellow
    Lamp1 (580,557 27x26), variable: Global.Tank1.Draining.State.Done, style: Lamp-Lamp1-Yellow
    Label (482,473 150x30), "DRAIN - PHASE"
    Label (397,588 53x30), "Running"
    Label (453,587 53x30), "Paused"
    Label (508,588 53x30), "Idle"
    Label (564,588 53x30), "Done"
    Button (714,640 58x30), "AUT"
        OnMouseClick: toggle Global.Tank1.Draining.Cmd.AutCtrl
    Button (713,524 58x30), "MAN"
        OnMouseClick: toggle Global.Tank1.Draining.Cmd.ManCtrl
    Lamp1 (733,688 27x26), variable: Global.Tank1.Draining.State.AutCtrl, style: Lamp-Lamp1-Yellow
    Lamp1 (733,570 27x26), variable: Global.Tank1.Draining.State.ManCtrl, style: Lamp-Lamp1-Yellow
    Button (384,523 58x30), "START"
        OnMouseClick: toggle Global.Tank1.Draining.Cmd.StartMan
    Button (451,523 58x30), "PAUSE"
        OnMouseClick: toggle Global.Tank1.Draining.Cmd.PauseMan
    Button (522,525 58x30), "STOP"
        OnMouseClick: toggle Global.Tank1.Draining.Cmd.StopMan
    Button (598,524 58x30), "RESUME"
        OnMouseClick: toggle Global.Tank1.Draining.Cmd.ResumeMan
    Button (383,640 58x30), "START"
        OnMouseClick: toggle Global.Tank1.Draining.Cmd.StartAut
    Button (513,640 58x30), "STOP"
        OnMouseClick: toggle Global.Tank1.Draining.Cmd.StopAut
    Lamp1 (395,681 27x26), variable: Global.Tank1.Draining.State.Running, style: Lamp-Lamp1-Yellow
    Lamp1 (531,679 27x26), variable: Global.Tank1.Draining.State.Idle, style: Lamp-Lamp1-Yellow
    Label (481,497 150x30), "MANUAL"
    Label (476,616 150x30), "AUTOMAT"
    Label (383,707 53x30), "Running"
    Label (518,705 53x30), "Idle"
    Label (723,241 53x30), "Manual"
    Label (719,591 53x30), "Manual"
    Label (722,358 53x30), "Automat"
    Label (718,709 53x30), "Automat"
    Rectangle (1094,159 125x156)
    Rectangle (1094,316 123x50)
    Rectangle (969,159 125x207)
    Rectangle (969,366 249x89)
    Button (1123,187 58x30), "AUT"
        OnMouseClick: toggle Global.Tank1.Mixer.Cmd.AutCtrl
    Button (995,185 58x30), "MAN"
        OnMouseClick: toggle Global.Tank1.Mixer.Cmd.ManCtrl
    Label (1000,135 212x18), "Mixer- Control moudule (CM)"
    Button (1015,277 58x30), "Open"
        OnMouseClick: toggle Global.Tank1.ValveFilling.Cmd.OpenMan
    Button (1015,310 58x30), "Close"
        OnMouseClick: toggle Global.Tank1.ValveFilling.Cmd.CloseMan
    Lamp1 (1139,225 27x26), variable: Global.Tank1.Mixer.State.AutCtrl, style: Lamp-Lamp1-Yellow
    Lamp1 (1012,230 27x26), variable: Global.Tank1.Mixer.State.ManCtrl, style: Lamp-Lamp1-Yellow
    Lamp1 (1003,406 27x26), variable: Global.Tank1.ValveFilling.State.Open, style: Lamp-Lamp1-Yellow
    Lamp1 (1079,406 27x26), variable: Global.Tank1.ValveFilling.State.Closed, style: Lamp-Lamp1-Yellow
    Lamp1 (1153,404 27x26), variable: Global.Tank1.ValveFilling.State.StartupFail, style: Lamp-Lamp1-Yellow
    Button (1124,327 58x30), "Res. SUF"
        OnMouseClick: toggle Global.Tank1.ValveFilling.Cmd.ResetSUF
    Label (986,378 53x18), "Opened"
    Label (1068,378 53x18), "Closed"
    Label (1152,380 33x18), "SUF"
    Lamp1 (972,277 27x26), variable: Global.Tank1.ValveFilling.State.OpenOut, style: Lamp-Lamp1-Yellow
    Lamp1 (972,311 27x26), variable: Global.Tank1.ValveFilling.State.CloseOut, style: Lamp-Lamp1-Yellow
END_VISUALIZATION
